Staubli VAL3: extAxisCan.pjx

--- extAxisCan.pjx ---
Parameters version=s7.6.3 stackSize=5000 millimeterUnit=true
Program file=CheckAxis.pgx
Program file=chkDrivesFault.pgx
Program file=chkDrivesOpEnab.pgx
Program file=chkDrivesSwOff.pgx
Program file=chkDrvState.pgx
Program file=chkLife.pgx
Program file=chkPosStatus.pgx
Program file=chkQuickStop.pgx
Program file=chkStatusWord.pgx
Program file=cmdAbortHoming.pgx
Program file=cmdDisableOp.pgx
Program file=cmdDisableVolt.pgx
Program file=cmdEnableHold.pgx
Program file=cmdEnableOp.pgx
Program file=cmdFaultReset.pgx
Program file=cmdQuickStop.pgx
Program file=cmdResetAll.pgx
Program file=cmdShutdown.pgx
Program file=cmdSwitchOn.pgx
Program file=getFbkPos.pgx
Program file=GoToPos.pgx
Program file=homing.pgx
Program file=init.pgx
Program file=IPMove.pgx
Program file=JogNegative.pgx
Program file=JogPositve.pgx
Program file=ReadMe.pgx
Program file=RecordExtAxis.pgx
Program file=RecordJoint.pgx
Program file=Reset.pgx
Program file=setCmdPos.pgx
Program file=setErrorCode.pgx
Program file=setHome.pgx
Program file=setOpMode.pgx
Program file=setPos.pgx
Program file=SingleMove.pgx
Program file=start.pgx
Program file=StepMove.pgx
Program file=stop.pgx
Program file=StopAll.pgx
Program file=stopExtAxis.pgx
Program file=Task4ms.pgx
Data file=extAxisCan.dtx
Library alias=cst path=Disk://constantes/constantes.pjx

--- extAxisCan.dtx ---
public aio aiPosFbk = {link=CanIO\Axis7\drvPosFbk_0}
public aio aoIPPos = {link=CanIO\Axis7\drvIPCmdPos_0}
public aio aoIPSpd = {link=CanIO\Axis7\ipVel_0}
public aio aoPosCmd = {link=CanIO\Axis7\drvCmdPos_0}
public aio aoWorkMode = {link=CanIO\Axis7\drvworkmode}
public bool bDriveQuickStop
public bool bDrivesOpEnable
bool bDrivesSwOnDis
public bool bDrvFault[2]
bool bEnableRequest
bool bIsS7_6 = true
bool bMemPower
public bool bNoDrivesFault = true
public bool bOpeEnabled[2]
bool bOverrun
public bool bQuickStop[2]
public bool bSWOnDis
public bool bSysShut
public bool blifebit[2]
  [0] = true
  [1] = true
bool blifebit_all_ok = true
public dio diFault = {link=CanIO\Axis7\fault_0}
public dio diHomingError = {link=CanIO\Axis7\homingError_0}
public dio diHomingReached = {link=CanIO\Axis7\homingReached_0}
public dio diIntLmtAct = {link=CanIO\Axis7\intLmtAct_0}
public dio diOpeEnabled = {link=CanIO\Axis7\opeEnabled_0}
public dio diPosReached = {link=CanIO\Axis7\targetReached_0}
public dio diQuickStop = {link=CanIO\Axis7\quickStopped_0}
public dio diReady2SwOn = {link=CanIO\Axis7\ready2SwOn_0}
public dio diSwOnDis = {link=CanIO\Axis7\swOnDis_0}
public dio diSwitchedOn = {link=CanIO\Axis7\switchedOn_0}
public dio diTargetReach = {link=CanIO\Axis7\targetReached_0}
public dio diVoltEnabled = {link=CanIO\Axis7\voltEnabled_0}
public dio diWarning = {link=CanIO\Axis7\warning_0}
public dio doEnableOp = {link=CanIO\Axis7\enableOp_0}
public dio doEnableVoltage = {link=CanIO\Axis7\enableVolt_0}
public dio doFaultReset = {link=CanIO\Axis7\faultReset_0}
public dio doManual = {link=CanIO\Axis7\Manual}
public dio doQuickStop = {link=CanIO\Axis7\quickStop_0}
public dio doStartHoming = {link=CanIO\Axis7\startHoming_0}
public dio doSwitchOn = {link=CanIO\Axis7\switchOn_0}
jointRx jDummy = {j1=1.48, j2=0.75, j3=2.04, j4=1.56, j5=2.81, j6=1.79}
jointRx jPosErrMax = {j1=100, j2=100, j3=100, j4=100, j5=100, j6=100}
jointRx jZero = {j1=0.01, j2=0.01, j3=0.01, j4=0.01, j5=0.01, j6=0.01}
public num nAxesPosFbk[2]
public num nAxesSum = 2
num nCntDrvDisable
num nCntDrvEnable[2]
public num nDrvFbkPos[2]
num nDrvPos[2]
num nDrvState[2]
  [0] = 1
  [1] = 1
public num nExtAxseAccDft = 10
public num nExtAxseSpdDft = 10
num nGearratio[2]
  [0] = 10
  [1] = 1
public num nResolution[2]
  [0] = 1280000
  [1] = 180000
public num nScaleFact[2]
  [0] = 10
  [1] = 360
public string sMsg
string sVersion = "s7.6 - May 29 2013 - 16:53:12"
public dio diRemote = {link=CanIO\Axis7\remote_0}
num nManul = 10
num nBuffSize
num nAxesData
public bool bMoveType
frame fFrame = {fatherId=world[0]}

--- start.pgx ---
program start()
  local num l_i
  local num l_sum
begin
  //
  call cst:init()
  call chkLife()
  if blifebit
    call init()
    taskCreateSync "T4ms",0.004,bOverrun,Task4ms()
  endIf
end

--- CheckAxis.pgx ---
public program CheckAxis(bool& x_b7Axis, bool& x_b8Axis)
begin

 x_b7Axis=$XgetNbAxes()>=1
 x_b8Axis=$XgetNbAxes()>=2


end

--- chkDrivesFault.pgx ---
program chkDrivesFault()
  local num l_i
begin
  //检查电机是否有错误
  //以下情况表明电机出现错误:
  //错误标志位；
  bNoDrivesFault=true
  for l_i=0 to nAxesSum-1
    if bDrvFault[l_i]!=(diFault[l_i]==true) and (!bDrvFault[l_i])
      sMsg="第"+toString("",l_i+1)+"轴控制器报错"
      popUpMsg(sMsg)
      logMsg(sMsg)
    endIf
    bDrvFault[l_i]=(diFault[l_i]==true)
    bNoDrivesFault=bNoDrivesFault and !bDrvFault[l_i]
  endFor
end

--- chkDrivesOpEnab.pgx ---
program chkDrivesOpEnab()
  local num l_i
begin
  //检查驱动器是否使能
  bDrivesOpEnable=true
  for l_i=0 to nAxesSum-1
    if  nDrvState[l_i]==5
      bOpeEnabled[l_i]=true
    else
      bOpeEnabled[l_i]=false
    endIf
    bDrivesOpEnable=bDrivesOpEnable and  bOpeEnabled[l_i]
  endFor

//
//  bDrivesOpEnable=bOpeEnabled[0]=(diOpeEnabled[0]==true and diSwitchedOn[0]==true and diQuickStop[0]==true )
//  for l_i=1 to nAxesSum-1
//    bOpeEnabled[l_i]=(diOpeEnabled[l_i]==true and diQuickStop[l_i]==true and  diSwitchedOn[l_i]==true )
//   // bOpeEnabled[l_i]=(diOpeEnabled[0]==true  and  diSwitchedOn[0]==true )
//    bDrivesOpEnable=bDrivesOpEnable and bOpeEnabled[l_i]
//  endFor
end

--- chkDrivesSwOff.pgx ---
program chkDrivesSwOff()
  local bool l_bDrvSwOnDis
  local num l_i
begin
  // 检测驱动器“switch on disabled"的状态
  bDrivesSwOnDis=true
  for l_i=0 to nAxesSum-1
    bSWOnDis[l_i]=(diSwOnDis[l_i]==true)
    bDrivesSwOnDis=bDrivesSwOnDis and bSWOnDis[l_i]
  endFor
  //
end

--- chkDrvState.pgx ---
program chkDrvState(num x_nAxisNum)
  local num l_nStatus
  local num l_nStatus1
  local bool l_bIsOneBitSet
begin
  //检查状态
  l_nStatus=0
  //确定电机是否在remote状态
  // read status_remote register
  //  call chkStatusRemote(x_nAxisNum,l_bIsOneBitSet)
  //  if l_bIsOneBitSet
  //    nDrvState[x_nAxisNum]=15
  //  else

  //读取状态字
  call chkStatusWord(x_nAxisNum,l_nStatus)
  //cst:nDRV_ACTIV:掩码，111dec=1101111bin.驱动器处于某种状态
  l_nStatus1=bAnd(l_nStatus,cst:nDRV_ACTIV)
  switch l_nStatus1
    //
    case cst:nRdy2SwitchON
      nDrvState[x_nAxisNum]=3
    break
    //
    case cst:nSwitchedON
      nDrvState[x_nAxisNum]=4
    break
    //使能
    case cst:nOperatEnabled
      nDrvState[x_nAxisNum]=5
    break
    //quickstop
    case cst:nQuickStopActiv
      nDrvState[x_nAxisNum]=12
    break
    //
    default
      //cst:nDRV_FAULT=100 1111
      l_nStatus1=bAnd(l_nStatus,cst:nDRV_FAULT)

      switch l_nStatus1
        case cst:nNotRdySwiON
          nDrvState[x_nAxisNum]=1
        break
        //
        case cst:nSwitchONDis
          nDrvState[x_nAxisNum]=2
        break
        //
        case cst:nFaultReacActiv
          nDrvState[x_nAxisNum]=13
        break
        //
        case cst:nFaultState
          nDrvState[x_nAxisNum]=14
        break
        //
        default
          nDrvState[x_nAxisNum]=-1
        break
      endSwitch
    break
    //
  endSwitch
end

--- chkLife.pgx ---
public program chkLife()
  local num l_i
  local string l_sMsg
begin
  //检查IO连接是否正常
  blifebit_all_ok=true
  for l_i=0 to nAxesSum-1
    if ioStatus(diReady2SwOn[l_i])<0
      blifebit[l_i]=false
      l_sMsg="第"+toString("",l_i+1)+"轴通讯异常"
      popUpMsg(l_sMsg)
      logMsg(l_sMsg)
      blifebit_all_ok=blifebit_all_ok and blifebit[l_i]
      return
    else
      blifebit[l_i]=true
      blifebit_all_ok=blifebit_all_ok and blifebit[l_i]
    endIf
  endFor

end

--- chkPosStatus.pgx ---
public program chkPosStatus(bool& x_bIsSame, num x_nAxisNum, num x_nAxisPos)
begin
  //检查外部轴是否在指定位置上
  x_bIsSame=abs(aioGet(aiPosFbk[x_nAxisNum])-x_nAxisPos*nGearratio[x_nAxisNum]*nResolution[x_nAxisNum]/nScaleFact[x_nAxisNum])<=5
end

--- chkQuickStop.pgx ---
program chkQuickStop()
  local num l_ni
begin
  //
  bDriveQuickStop=false
  for l_ni=0 to nAxesSum-1
    if nDrvState[l_ni]==12
      bQuickStop[l_ni]=true
    else
      bQuickStop[l_ni]=false
    endIf
    bDriveQuickStop=bDriveQuickStop or bQuickStop[l_ni]
  endFor
end

--- chkStatusWord.pgx ---
program chkStatusWord(num x_nAxisNumber, num& x_nValue)
begin
  //返回电机状态字的数值
  //  x_nValue=aioGet(aiStatusWord[x_nAxisNumber])
  x_nValue=dioGet(diReady2SwOn[x_nAxisNumber])*power(2,0)
  x_nValue=dioGet(diSwitchedOn[x_nAxisNumber])*power(2,1)+x_nValue
  x_nValue=dioGet(diOpeEnabled[x_nAxisNumber])*power(2,2)+x_nValue
  x_nValue=dioGet(diFault[x_nAxisNumber])*power(2,3)+x_nValue
  x_nValue=dioGet(diVoltEnabled[x_nAxisNumber])*power(2,4)+x_nValue
  x_nValue=dioGet(diQuickStop[x_nAxisNumber])*power(2,5)+x_nValue
  x_nValue=dioGet(diSwOnDis[x_nAxisNumber])*power(2,6)+x_nValue
  x_nValue=dioGet(diWarning[x_nAxisNumber])*power(2,7)+x_nValue
  x_nValue=dioGet(diRemote[x_nAxisNumber])*power(2,9)+x_nValue
  x_nValue=dioGet(diTargetReach[x_nAxisNumber])*power(2,10)+x_nValue
  x_nValue=dioGet(diIntLmtAct[x_nAxisNumber])*power(2,11)+x_nValue
  x_nValue=dioGet(diHomingReached[x_nAxisNumber])*power(2,12)+x_nValue
  x_nValue=dioGet(diHomingError[x_nAxisNumber])*power(2,13)+x_nValue
end

--- cmdAbortHoming.pgx ---
public program cmdAbortHoming(num x_nAxisNum)
begin
 //取消回零

end

--- cmdDisableOp.pgx ---
public program cmdDisableOp(num x_nAxNum)
begin
  //发送“终止操作”指令到所选驱动器
  if bOpeEnabled[x_nAxNum]==true
    doFaultReset[x_nAxNum]=false
    doEnableOp[x_nAxNum]=false
    delay(0.1)
    doQuickStop[x_nAxNum]=true
    doEnableVoltage[x_nAxNum]=true
    doSwitchOn[x_nAxNum]=true
  endIf
end

--- cmdDisableVolt.pgx ---
public program cmdDisableVolt(num x_nAxNum)
begin
  //"Disable voltage"字段无效
  doFaultReset[x_nAxNum]=false
  doEnableVoltage[x_nAxNum]=false
end

--- cmdEnableHold.pgx ---
public program cmdEnableHold(num x_nAxNum (dimensions=1))
begin
  // this program issues an 'Enable Hold'  command to the selected drive.
  // This bit must be set to enable drive power
  //发送“enable hold”指令到所选控制器
  //用于设置驱动器电源开启
  //  doEnableHold[x_nAxNum]=true
end

--- cmdEnableOp.pgx ---
public program cmdEnableOp(num x_nAxNum)
begin
  //设置'Enable Operation'
  if bOpeEnabled[x_nAxNum]==false
    doFaultReset[x_nAxNum]=false
    doSwitchOn[x_nAxNum]=false
    doEnableOp[x_nAxNum]=false
    doEnableVoltage[x_nAxNum]=true
    doQuickStop[x_nAxNum]=true
    delay(0.1)
    doSwitchOn[x_nAxNum]=true
    delay(0.1)
    doEnableOp[x_nAxNum]=true
    delay(0.1)
  endIf
end

--- cmdFaultReset.pgx ---
public program cmdFaultReset(num x_nAxNum)
begin
  //错误复位，'Fault reset'置1
  doFaultReset[x_nAxNum]=true
  delay(0.008)
  doFaultReset[x_nAxNum]=false
end

--- cmdQuickStop.pgx ---
public program cmdQuickStop(num x_nAxNum)
begin
  //"quickstop"置为false
  //激活quickstop
  if !bQuickStop[x_nAxNum]
    doFaultReset[x_nAxNum]=false
    doEnableVoltage[x_nAxNum]=true
    doSwitchOn[x_nAxNum]=true
    doEnableOp[x_nAxNum]=true
    delay(0.1)
    doQuickStop[x_nAxNum]=false
    delay(0.1)
  endIf
end

--- cmdResetAll.pgx ---
public program cmdResetAll(num x_nAxNum)
begin
  //复位所有信号
  doFaultReset[x_nAxNum]=false
  doEnableOp[x_nAxNum]=false
  doSwitchOn[x_nAxNum]=false
  doEnableVoltage[x_nAxNum]=false
  doQuickStop[x_nAxNum]=false
  delay(0.1)
end

--- cmdShutdown.pgx ---
public program cmdShutdown(num& x_nAxNum)
begin
  //关闭指定驱动器，设置"switch on"为false
  //shutdown的顺序参考相应电机说明
  doFaultReset[x_nAxNum]=false
  doQuickStop[x_nAxNum]=true
  doEnableVoltage[x_nAxNum]=true
  doSwitchOn[x_nAxNum]=false
  delay(0.004)
end

--- cmdSwitchOn.pgx ---
public program cmdSwitchOn(num& x_nAxNum)
begin
  //"switch on"设置为true
  doFaultReset[x_nAxNum]=false
  doEnableOp[x_nAxNum]=false
  doQuickStop[x_nAxNum]=true
  doEnableVoltage[x_nAxNum]=true
  doSwitchOn[x_nAxNum]=true
  delay(0.1)
end

--- DAEMON1.PGX ---
public program daemon1()
  local num l_nKey
begin

  while (getKey()!=270)
    call daemon4()
    delay(0)
  endWhile
end

--- DAEMON2.PGX ---
public program daemon2()
  local jointRx l_jCurr
  local num l_i
  local bool l_bError
  local string l_sMsg
  local num l_nError
  local bool l_bDrivesOK
begin

  // Verification du bit de vie bus can
  call chkLifeBit()

  // Gestion watchDog pour variateurs
  //call updateWatchDog()
  //
  // Recupere etat des variateurs
  l_bDrivesOK=true
  for l_i=0 to nNUMOFAXES-1
    bDrvFault[l_i]=(diFault[l_i]==true) or bAnd(aioGet(aiStatusRemote[l_i])/32,255)!=0
    call chkDrvState(l_i)
    l_bDrivesOK=l_bDrivesOK and nDrvState[l_i]==cst:nOperatEnabled
    bDrivesOpEnable=l_bDrivesOK
  endFor

  if isPowered() and l_bDrivesOK
    // Get system position
    $XgetDrvCmdPos(nDrvPos)
    l_sMsg=""
    //$XgetJntCmdPos(l_nJntPos)
    for l_i=0 to nNUMOFAXES-1
      // Send it to the external axis
      aioSet(aoPosCmd[l_i],nDrvPos[l_i]*nScaleFact)
      //l_sMsg="0: "+toString(".3",l_nJntPos[0])+"   1: "+toString(".3",l_nJntPos[1])
      l_sMsg=l_sMsg+toString("",l_i)+": "+toString(".3",nDrvPos[l_i])+"   "
    endFor
    //? l_sMsg
  else
    for l_i=0 to nNUMOFAXES-1
      doEnableOp[l_i]=false
      doSwitchOn[l_i]=false
      // Get external axis position
      nDrvPos[l_i]=aioGet(aiPosFbk[l_i])/nScaleFact
    endFor
    // Update it in the system
    $XsetDrvFbkPos(nDrvPos)
  endIf



end

--- getFbkPos.pgx ---
public program getFbkPos()
  local num l_i
begin
  for l_i=0 to nAxesSum-1
      //nScaleFact:电机转一圈角度（旋转轴）或前进距离（直线轴（mm））
      nDrvFbkPos[l_i]=nScaleFact[l_i]*aioGet(aiPosFbk[l_i])/nResolution[l_i]*nGearratio[l_i]
      nAxesPosFbk[l_i]=nDrvFbkPos[l_i]/nGearratio[l_i]
  endFor
end

--- getStatusWord.pgx ---
public program getStatusWord(num x_nAxisNumber, num& x_nValue)
begin
  // this routine return the value of the drive's status word
  //
  x_nValue=aioGet(aiStatusWord[x_nAxisNumber])
end

--- GoToPos.pgx ---
public program GoToPos(num x_nAxisNum, num x_nPos)
begin

  if !isPowered()
    popUpMsg("请先给机器人上电")
    return
  endIf
  doStartHoming[x_nAxisNum]=false
  aioSet(aoWorkMode[x_nAxisNum],cst:nPPMODE)
  delay(0.1)
  aioSet(aoPosCmd[x_nAxisNum],x_nPos*nResolution[x_nAxisNum]/nScaleFact[x_nAxisNum])
  delay(0.1)
  doStartHoming[x_nAxisNum]=true
  doManual[x_nAxisNum]=true
  wait(diTargetReach[x_nAxisNum]==false)
  wait(diTargetReach[x_nAxisNum]==true)
  disablePower()
  delay(0.1)
  aioSet(aoWorkMode[x_nAxisNum],cst:nINTERPMODE)
  doStartHoming[x_nAxisNum]=true
end

--- homing.pgx ---
public program homing(num x_nAxisNum, bool& x_bRes)
  local bool l_bError
  local num l_nEtape
  local string l_sMsg
  local num l_nTps
  local bool l_bVerrou
  local bool l_bOK
  local num l_nDuration
  local string l_sYN[2]
  local num l_nDrvPos
begin
  //指定外部轴零点
  //  if !isPowered()
  //    popUpMsg("请先上电")
  //    return
  //  endIf
  //  x_bRes=false
  //  doStartHoming[x_nAxisNum]=false
  //  delay(0.1)
  //  aioSet(aoWorkMode[x_nAxisNum],6)
  //  doStartHoming[x_nAxisNum]=true
  //  l_sYN[0]="是"
  //  l_sYN[1]="否"
  //  if watch(diHomingReached[x_nAxisNum]==true,2)
  //    x_bRes=true
  //    popUpMsg("设置成功")
  //  endIf

  //
  x_bRes=false
  if !isPowered()
    popUpMsg("请先给机器人上电")
    return
  endIf
  doStartHoming[x_nAxisNum]=false
  aioSet(aoWorkMode[x_nAxisNum],cst:nHOMINGMODE)
  delay(0.1)
  doStartHoming[x_nAxisNum]=true
  wait(diHomingReached[x_nAxisNum]==false)
  wait(diHomingReached[x_nAxisNum]==true)
  disablePower()
  delay(0.1)
  aioSet(aoWorkMode[x_nAxisNum],cst:nINTERPMODE)
  x_bRes=true
end

--- init.pgx ---
public program init()
  local num l_i
  local bool l_bError
begin

  call cst:init()
  //获取外部轴数目
  nAxesSum=$XgetNbAxes()

  if nAxesSum<1
    popUpMsg("外部轴不正确")
    return
  endIf

  //根据外部轴数目更改变量数目
  resize(nCntDrvEnable,1,nAxesSum)
  resize(nDrvPos,1,nAxesSum)
  resize(bDrvFault,1,nAxesSum)
  resize(nAxesPosFbk,1,nAxesSum)
  resize(nDrvFbkPos,1,nAxesSum)
  resize(bDrvFault,1,nAxesSum)
  resize(bOpeEnabled,1,nAxesSum)
  resize(bQuickStop,1,nAxesSum)
  resize(blifebit,1,nAxesSum)
  resize(nDrvState,1,nAxesSum)
  //  if size(nDrvPos)!=nAxesSum
  //    resize(nDrvPos,1,nAxesSum)
  //  endIf

  //  if size(nDrvFbkPos)!=nAxesSum
  //    resize(nDrvFbkPos,1,nAxesSum)
  //  endIf
  //  if size(bDrvFault)!=nAxesSum
  //    resize(bDrvFault,1,nAxesSum)
  //  endIf
  //  if size(nAxesPosFbk)!=nAxesSum
  //    resize(nAxesPosFbk,1,nAxesSum)
  //  endIf
  //  if size(bOpeEnabled)!=nAxesSum
  //    resize(bOpeEnabled,1,nAxesSum)
  //  endIf
  //
  //  if size(bQuickStop)!=nAxesSum
  //    resize(bQuickStop,1,nAxesSum)
  //  endIf
  //
  //  if size(blifebit)!=nAxesSum
  //    resize(blifebit,1,nAxesSum)
  //  endIf
  //
  //  if size(nCntDrvEnable)!=nAxesSum
  //    resize(nCntDrvEnable,1,nAxesSum)
  //  endIf
  //
  //  // 驱动器状态变量
  //  if size(nDrvState)!=nAxesSum
  //    resize(nDrvState,1,nAxesSum)
  //  endIf
  //
  //





  //初始化
  for l_i=0 to nAxesSum-1
    call cmdResetAll(l_i)
    call cmdFaultReset(l_i)
    bDrvFault[l_i]=false
    aioSet(aoWorkMode[l_i],cst:nINTERPMODE)
    doStartHoming[l_i]=true
    nCntDrvEnable[l_i]=0
    bQuickStop=false
  endFor
  delay(0.008)
  disablePower()
  wait(isPowered()==false)
  bSysShut=false
  //
  // call Version()
  // libSave()
end

--- IPMove.pgx ---
public program IPMove()
begin
  //
//  $XgetDrvCmdPos(nDrvPos)
//  for l_i=0 to nAxesSum-1
//    aioSet(aoIPPos[l_i],(nDrvPos[l_i]*nResolution[l_i]/nScaleFact[l_i]))
//  endFor
end

--- JogNegative.pgx ---
public program JogNegative(num x_nAxis, num x_nKey)
begin
  call StepMove(x_nAxis,x_nKey,false)
end

--- JogPositve.pgx ---
public program JogPositve(num x_nAxis, num x_nKey)
begin
  call StepMove(x_nAxis,x_nKey,true)
end

--- pwrOffDrive1.pgx ---
public program pwrOffDrive1(num x_nAxNum, num& x_nError)
  local bool l_bVerrou
  local num l_nEtape
  local bool l_bOK
  local string l_sMsg
  local num l_nMemEtape
  local bool l_bQuit
begin

  l_bVerrou=false
  l_nMemEtape=-1
  l_bQuit=false
  x_nError=0

  // sequenceur pour desactiver les variateurs
  while !l_bQuit
    // Read current drive State
    //call getDriveState(x_nAxNum,nDrvState[x_nAxNum])
    l_nEtape=nDrvState[x_nAxNum]
    // Changement d'état ?
    if l_nEtape!=l_nMemEtape
      l_nMemEtape=l_nEtape
      l_bVerrou=false
    endIf

    l_sMsg="pwrOffDrive>>Etape : "+toString("",l_nEtape)+" "
    switch l_nEtape
      // Not ready to Switch on
      case 1
        if l_bVerrou==false
          if bAnd(nDebug,cst:nDEBUGDRIVE)==cst:nDEBUGDRIVE
            l_sMsg=l_sMsg+"Not ready to Switch on"
            logMsg(l_sMsg)
          endIf
          l_bVerrou=true
        endIf
      break
      // Switch ON disabled
      case 2
        if l_bVerrou==false
          if bAnd(nDebug,cst:nDEBUGDRIVE)==cst:nDEBUGDRIVE
            l_sMsg=l_sMsg+"Switch on disabled"
            logMsg(l_sMsg)
          endIf
          l_bQuit=true
          call cmdResetAll(x_nAxNum)
          l_bVerrou=true
        endIf
      break
      // Ready to switch on
      case 3
        if l_bVerrou==false
          if bAnd(nDebug,cst:nDEBUGDRIVE)==cst:nDEBUGDRIVE
            l_sMsg=l_sMsg+"Ready to switch on"
            logMsg(l_sMsg)
          endIf
          call cmdQuickStop(x_nAxNum)
          call cmdDisableVolt(x_nAxNum)
          l_bVerrou=true
        endIf
      break
      // Switched ON
      case 4
        if l_bVerrou==false
          if bAnd(nDebug,cst:nDEBUGDRIVE)==cst:nDEBUGDRIVE
            l_sMsg=l_sMsg+"Switched ON"
            logMsg(l_sMsg)
          endIf
          //          call cmdQuickStop(x_nAxNum)
          //          call cmdDisableVolt(x_nAxNum)
          //
          call cmdShutdown(x_nAxNum)
          l_bVerrou=true
        endIf
      break
      // Operation enabled
      case 5
        if l_bVerrou==false
          if bAnd(nDebug,cst:nDEBUGDRIVE)==cst:nDEBUGDRIVE
            l_sMsg=l_sMsg+"Operation enabled"
            logMsg(l_sMsg)
          endIf
          //          call cmdDisableVolt(x_nAxNum)

          //*******
          call cmdDisableOp(x_nAxNum)
          // ******
          l_bVerrou=true
        endIf
      break

      // Fault state
      case 14
        if l_bVerrou==false
          if bAnd(nDebug,cst:nDEBUGDRIVE)==cst:nDEBUGDRIVE
            l_sMsg=l_sMsg+"Fault state"
            logMsg(l_sMsg)
          endIf
          l_bQuit=true
          x_nError=1
          l_bVerrou=true
        endIf
      break
      //
      // Alarm from status_remote register is set
      case 15
        if l_bVerrou==false
          if bAnd(nDebug,cst:nDEBUGDRIVE)==cst:nDEBUGDRIVE
            l_sMsg=l_sMsg+"Alarm Status_remote register"
            logMsg(l_sMsg)
          endIf
          l_bQuit=true
          x_nError=2
          call cmdResetAll(x_nAxNum)
          l_bVerrou=true
        endIf
      break
      //
    endSwitch
    delay(0)
  endWhile

end

--- pwrOffDrive2.pgx ---
public program pwrOffDrive2(num x_nAxNum)
  local bool l_bOK
  local string l_sMsg
begin
  // sequenceur pour desactiver les variateurs

  // Read current drive State
  call chkDrvState(x_nAxNum)

  // Changement d'état ?
  if nDrvState[x_nAxNum]!=nMemPwrOffStep[x_nAxNum]
    nMemPwrOffStep[x_nAxNum]=nDrvState[x_nAxNum]
    bLockPwrOff[x_nAxNum]=false
  endIf

  l_sMsg="pwrOffDrive>>Etape : "+toString("",nDrvState[x_nAxNum])+" "
  switch nDrvState[x_nAxNum]
    // Not ready to Switch on
    case 1
      if bLockPwrOff[x_nAxNum]==false
        if bAnd(nDebug,cst:nDEBUGDRIVE)==cst:nDEBUGDRIVE
          l_sMsg=l_sMsg+"Not ready to Switch on"
          logMsg(l_sMsg)
        endIf
        bLockPwrOff[x_nAxNum]=true
      endIf
    break
    // Switch ON disabled
    case 2
      if bLockPwrOff[x_nAxNum]==false
        if bAnd(nDebug,cst:nDEBUGDRIVE)==cst:nDEBUGDRIVE
          l_sMsg=l_sMsg+"Switch on disabled"
          logMsg(l_sMsg)
        endIf
        call cmdResetAll(x_nAxNum)
        bLockPwrOff[x_nAxNum]=true
      endIf
    break
    // Ready to switch on
    case 3
      if bLockPwrOff[x_nAxNum]==false
        if bAnd(nDebug,cst:nDEBUGDRIVE)==cst:nDEBUGDRIVE
          l_sMsg=l_sMsg+"Ready to switch on"
          logMsg(l_sMsg)
        endIf
        call cmdQuickStop(x_nAxNum)
        call cmdDisableVolt(x_nAxNum)
        bLockPwrOff[x_nAxNum]=true
      endIf
    break
    // Switched ON
    case 4
      if bLockPwrOff[x_nAxNum]==false
        if bAnd(nDebug,cst:nDEBUGDRIVE)==cst:nDEBUGDRIVE
          l_sMsg=l_sMsg+"Switched ON"
          logMsg(l_sMsg)
        endIf
        call cmdShutdown(x_nAxNum)
        bLockPwrOff[x_nAxNum]=true
      endIf
    break
    // Operation enabled
    case 5
      if bLockPwrOff[x_nAxNum]==false
        if bAnd(nDebug,cst:nDEBUGDRIVE)==cst:nDEBUGDRIVE
          l_sMsg=l_sMsg+"Operation enabled"
          logMsg(l_sMsg)
        endIf
        call cmdDisableOp(x_nAxNum)
        bLockPwrOff[x_nAxNum]=true
      endIf
    break

    // Fault state
    case 14
      if bLockPwrOff[x_nAxNum]==false
        if bAnd(nDebug,cst:nDEBUGDRIVE)==cst:nDEBUGDRIVE
          l_sMsg=l_sMsg+"Fault state"
          logMsg(l_sMsg)
        endIf
        bLockPwrOff[x_nAxNum]=true
      endIf
    break
    //
    // Alarm from status_remote register is set
    case 15
      if bLockPwrOff[x_nAxNum]==false
        if bAnd(nDebug,cst:nDEBUGDRIVE)==cst:nDEBUGDRIVE
          l_sMsg=l_sMsg+"Alarm Status_remote register"
          logMsg(l_sMsg)
        endIf
        call cmdResetAll(x_nAxNum)
        bLockPwrOff[x_nAxNum]=true
      endIf
    break
    //
  endSwitch

end

--- pwrOffDrives.pgx ---
public program pwrOffDrives()
  local num l_i
begin
  for l_i=0 to nNUMOFAXES-1
    doEnableVoltage[l_i]=false
    doQuickStop[l_i]=false
    doSwitchOn[l_i]=false
    doEnableOp[l_i]=false
  endFor
end

--- ReadMe.pgx ---
program ReadMe()
begin
//在通用版本上对lasman进行定制
//1.添加了三个四个函数
//checkAxis
//SingleMove
//RecordExtAxis
//RecordJoint


//还有一些变量需要添加







end

--- RecordExtAxis.pgx ---
public program RecordExtAxis(trsf& x_trTrsf, trsf& x_trPos, tool x_tTool)
  local jointRx l_jJ
  local pointRx l_pP
begin
  //  $recClean("c")
  //  $recAdd("c","CanIO\Axis8\posCmd_1")
  //  $recAdd("c","CanIO\Axis8\posFbk_1")
  //  $recStart("c",50,250)

  //  $recClean("c")
  //  $recAdd("c","extDrvCmdPos")
  //  $recAdd("c","extDrvCmdVel")
  //  $recAdd("c","extJntCmdPos")
  //  $recAdd("c","extJntCmdVel")
  //  $recAdd("c","extError")
  //  $recAdd("c","extDrvGrpError")
  //  $recStart("c",50,250)

 // x_pPos=$here
//    resize(nBuffSize,1,sel(x_b8Axis,2,1))
//  x_j=$XH(nBuffSize)
//  x_trTrsf.x=nBuffSize[0]
//  if x_b8Axis
//    x_trTrsf.y=nBuffSize[1]
//  endIf


if bMoveType
  $XframeLink(fFrame)
 l_pP=here(x_tTool,fFrame)
  x_trPos=l_pP.trsf

endIf




//记录七轴，八轴位置
call RecordJoint(l_jJ,x_trTrsf)




end

--- RecordJoint.pgx ---
public program RecordJoint(jointRx& x_j, trsf& x_trTrsf)
  local num l_nNum[2]
begin
  //  $recClean("c")
  //  $recAdd("c","CanIO\Axis8\posCmd_1")
  //  $recAdd("c","CanIO\Axis8\posFbk_1")
  //  $recStart("c",50,250)

  //  $recClean("c")
  //  $recAdd("c","extDrvCmdPos")
  //  $recAdd("c","extDrvCmdVel")
  //  $recAdd("c","extJntCmdPos")
  //  $recAdd("c","extJntCmdVel")
  //  $recAdd("c","extError")
  //  $recAdd("c","extDrvGrpError")
  //  $recStart("c",50,250)

 // x_pPos=$here

 //记录轴的值
  if nAxesSum<1
    popUpMsg("轴个数错误")
    return
  endIf

  resize(nBuffSize,1,nAxesSum)
  x_j=$Xherej(nBuffSize)
  x_trTrsf.x=nBuffSize[0]
  if nAxesSum>1
    x_trTrsf.y=nBuffSize[1]
  endIf

end

--- Reset.pgx ---
public program Reset()
  local num l_i
begin
  //报警复位
  for l_i=0 to nAxesSum-1
    call cmdFaultReset(l_i)
  endFor
//  call user:timerDialog("复位完成",0.5)
end

--- setCmdPos.pgx ---
program setCmdPos(num x_nAxisNum (dimensions=1))
  local num l_nCurrentPos
  local num l_nCmdPos
begin
  //把当前位置赋给驱动器
  l_nCurrentPos=aioGet(aiPosFbk[x_nAxisNum])
  aioSet(aoPosCmd[x_nAxisNum],l_nCurrentPos)
end

--- setErrorCode.pgx ---
program setErrorCode(num x_nAxisNum (dimensions=1), num& x_nErrorCode (dimensions=1))
  local num l_nAlarm
begin
  // This program returns the value of the current error
  //获取当前错误代码值
  x_nErrorCode=0
  //检查电机错误位是否被设置
  // Check if driveFault bit is set
  //  if diFault[x_nAxisNum]==true
  //    //硬件错误
  //    // Hardware alarm ?
  //    call chkHwAlarm(x_nAxisNum,x_nErrorCode)
  //    if x_nErrorCode==0
  //      // Software alarm ?
  //      call chkSwAlarm(x_nAxisNum,x_nErrorCode)
  //    endIf
  //    // Check alarm bits of status_remote register
  //  elseIf nAppV3Error[x_nAxisNum]==0
  //    call getRegisterVal(cst:nSTATUS_REMOTE,x_nAxisNum,x_nErrorCode)
  //  else
  //    // Check if Application error
  //    x_nErrorCode=nAppV3Error[x_nAxisNum]
  //  endIf
end

--- setHome.pgx ---
public program setHome(num x_nAxisNum, bool& x_bRes)
  local bool l_bError
  local num l_nEtape
  local string l_sMsg
  local num l_nTps
  local bool l_bVerrou
  local bool l_bOK
  local num l_nDuration
  local string l_sYN[2]
  local num l_nDrvPos
begin
  //对绝对编码器电机设置当前值位为零点
    if !isPowered()
      popUpMsg("请先上电")
      return
    endIf
    x_bRes=false
    doStartHoming[x_nAxisNum]=false
    delay(0.1)
    aioSet(aoWorkMode[x_nAxisNum],cst:nHOMINGMODE)
    doStartHoming[x_nAxisNum]=true
    wait(diHomingReached[x_nAxisNum]==false)
    wait(diHomingReached[x_nAxisNum]==true)
    if watch(diHomingReached[x_nAxisNum]==true,2)
      x_bRes=true
      popUpMsg("设置成功")
    endIf
    disablePower()
    delay(0.008)
    aioSet(aoWorkMode[x_nAxisNum],cst:nINTERPMODE)
 end

--- setOpMode.pgx ---
public program setOpMode(num x_nAxisNum, num x_nOpMode)
  local num l_nK
begin

  //call checkDin(diSwitchedOn[x_nAxisNum],false,x_bError)

  // Interpolated position mode
  //  aioSet(aoMoop[x_nAxisNum],x_nOpMode)
  aioSet(aoWorkMode[x_nAxisNum],x_nOpMode)
  // Reset fault
//  doFaultReset[x_nAxisNum]=false
//  delay(0.1)
//  doFaultReset[x_nAxisNum]=true
//  delay(0.1)
//  doFaultReset[x_nAxisNum]=false

  // Copy current axis position into commanded position
  // Probably not necessary need to be checked.
  //  call setCmdPos(x_nAxisNum)

  //  // Init watchdog
  //  doEnableHold[x_nAxisNum]=true
  //  doWatchDog[x_nAxisNum]=true
  //  // Starting sequence
  //  doEnableVoltage[x_nAxisNum]=true
  //  doQuickStop[x_nAxisNum]=true

  //call checkDin(diReady2SwOn[x_nAxisNum],true,x_bError)


end

--- setPos.pgx ---
program setPos(num x_nAxisNum (dimensions=1), num x_nCurrentPos (dimensions=1))
begin
  //
  aioSet(aoPosCmd[x_nAxisNum],x_nCurrentPos)
end

--- SingleMove.pgx ---
public program SingleMove(num x_nType, jointRx x_j, pointRx x_pM, pointRx x_pE, tool x_tTool, mdesc x_m, trsf x_trExtAxis)
  local pointRx l_pP[2]
begin
  if x_nType<1 or x_nType>3
    return
  endIf

  resize(nAxesData,1,nAxesSum)
  nAxesData[0]=x_trExtAxis.x
  if nAxesSum>=2
    nAxesData[1]=x_trExtAxis.y

  endIf



  if !bMoveType or x_nType==1

    switch x_nType
      case 1
        $Xmovej(x_j,nAxesData,x_tTool,x_m)
      break


      case 2
        $Xmovel(x_pE,nAxesData,x_tTool,x_m)
      break

      case 3
        $Xmovec(x_pM,x_pE,nAxesData,x_tTool,x_m)
      break


    endSwitch
    return


  endIf





  //2014.12.04
  //对于离线进行修改
  //fFrame.trsf={0,0,0,0,0,0}
  if bMoveType
    $XframeLink(fFrame)
  else
    link(fFrame,world)
  endIf





  link(l_pP[0],fFrame)
  link(l_pP[1],fFrame)


  l_pP[0].trsf=x_pM.trsf
  l_pP[1].trsf=x_pE.trsf

  //×××××××××××××××××××××××××××××××××××××××××××
  switch x_nType
    case 1
      $Xmovej(x_j,nAxesData,x_tTool,x_m)
    break

    case 2
      $Xmovel(l_pP[1],nAxesData,x_tTool,x_m)
    break

    case 3
      $Xmovec(l_pP[0],l_pP[1],nAxesData,x_tTool,x_m)
    break

  endSwitch


end

--- StepMove.pgx ---
public program StepMove(num x_nAxisNum, num x_nKey, bool x_bJog)
begin
  //
  if isKeyPressed(x_nKey)
    //x_bjog=true:正向运动
    if x_bJog
      ? "+"
      aioSet(aoWorkMode[x_nAxisNum],-1)
      doStartHoming[x_nAxisNum]=true
    else
      ? "-"
      aioSet(aoWorkMode[x_nAxisNum],-1)
      doManual[x_nAxisNum]=true
    endIf
    wait(isKeyPressed(x_nKey)==false)
  else
    doStartHoming[x_nAxisNum]=false
    doManual[x_nAxisNum]=false
  endIf
end

--- stop.pgx ---
public program stop()
  local num l_i
begin
  call StopAll()


end

--- StopAll.pgx ---
public program StopAll()
  local num l_ni
begin
  for l_ni=0 to nAxesSum-1
    call stopExtAxis(l_ni)
  endFor
end

--- stopExtAxis.pgx ---
public program stopExtAxis(num x_nAxisNum)
begin
  //
  if blifebit[x_nAxisNum]
    doQuickStop[x_nAxisNum]=false
    doSwitchOn[x_nAxisNum]=false
    doEnableVoltage[x_nAxisNum]=false
    doEnableOp[x_nAxisNum]=false
    doStartHoming[x_nAxisNum]=false
    aioSet(aoWorkMode[x_nAxisNum],0)
  endIf
end

--- SYNCMOVE.pgx ---
public program syncMove(num& x_nAxisNum[])
  local jointRx l_jCurr
  local num l_nEncRes
  local num l_nDrvPos[2]
  local bool l_bFirstRun
  local num l_i
  local bool l_bError
  local string l_sMsg
begin

  l_nEncRes=8192/360

  call setCmdPos(0)
  call setCmdPos(1)
  bStop=false
  l_bFirstRun=true

  // Ne pas supprimer ces lignes
  disablePower()
  wait(isPowered()==false)
  //wait(isPowered()==true)
  /// FIN /////////////

  while !bStop
    if (isPowered()==true) and (l_bFirstRun==false)
      for l_i=0 to size(x_nAxisNum)-1
        if (diSwitchedOn[x_nAxisNum[l_i]]==false)
          doSwitchOn[x_nAxisNum[l_i]]=true
          delay(0.05)
          doEnableOp[x_nAxisNum[l_i]]=true
        endIf
      endFor
      // Get system position
      $XgetDrvCmdPos(l_nDrvPos)
      //$XgetJntCmdPos(l_nJntPos)
      // Send it to the external axis
      aioSet(aoPosCmd[x_nAxisNum[0]],l_nDrvPos[0]*l_nEncRes)
      aioSet(aoPosCmd[x_nAxisNum[1]],l_nDrvPos[1]*l_nEncRes)
      //l_sMsg="0: "+toString(".3",l_nJntPos[0])+"   1: "+toString(".3",l_nJntPos[1])
      l_sMsg="0: "+toString(".3",l_nDrvPos[0])+"   1: "+toString(".3",l_nDrvPos[1])
      //? l_sMsg
    else
      for l_i=0 to size(x_nAxisNum)-1
        doSwitchOn[x_nAxisNum[l_i]]=false
        doEnableOp[x_nAxisNum[l_i]]=false
      endFor
      // Get external axis position
      l_nDrvPos[0]=aioGet(aiPosFbk[x_nAxisNum[0]])/l_nEncRes
      l_nDrvPos[1]=aioGet(aiPosFbk[x_nAxisNum[1]])/l_nEncRes
      // Update it in the system
      $XsetDrvFbkPos(l_nDrvPos)
    endIf
    delay(0)
    l_bFirstRun=false
  endWhile
end

--- Task4ms.pgx ---
public program Task4ms()
  local num l_i
  local num l_nWorking
  local num l_nStatus
begin
  //4ms的任务,检测外部轴的状态信息
  while true
    //检查通讯是否正常
    call chkLife()
    if !blifebit_all_ok
      resetMotion()
      stopMove()
      disablePower()
      popUpMsg("同步外部轴异常")
      bSysShut=true
      return
    endIf
    //检查错误
    call chkDrivesFault()
    //检查状态
    for l_i=0 to nAxesSum-1
      call chkDrvState(l_i)
    endFor
    //反馈位置
    call getFbkPos()
    // 检查所有驱动器是否在operation enabled
    call chkDrivesOpEnab()
    //检测quickstop
    call chkQuickStop()
    //s7.6以上版本


    //使用在s7.5及以下系统时，命令行注释
    bEnableRequest=isPowered()
    //使用在s7.6，命令行注释
    $XdrvEnable(bEnableRequest,bDrivesOpEnable)
    //
    if bEnableRequest
      if bMemPower==false
        // 触发使能次数
        for l_i=0 to nAxesSum-1
          nCntDrvEnable[l_i]=0
        endFor
        bMemPower=true
      endIf
      //
      if bNoDrivesFault
        if bDrivesOpEnable
          //从$XMovel,$XMovej和$XMovec指令中获得外部轴离散位置(4ms的距离)
          $XgetDrvCmdPos(nDrvPos)
          for l_i=0 to nAxesSum-1
            aioSet(aoIPPos[l_i],(nDrvPos[l_i]/nGearratio[l_i]*nResolution[l_i]/nScaleFact[l_i]))
          endFor
          bSysShut=false
        else
          //增加触发使能次数
          l_i=0
          for l_i=0 to nAxesSum-1
            if bOpeEnabled==false
              // cst:nTO_DRVDISABLE=2
              if nCntDrvEnable[l_i]<250*cst:nTO_DRVDISABLE
                call cmdEnableOp(l_i)
              else
                sMsg="轴"+toString("",l_i+7)+"使能超时"
                popUpMsg(sMsg)
                logMsg(sMsg)
                bSysShut=true
                disablePower()
                return
              endIf
            endIf
            nCntDrvEnable[l_i]=nCntDrvEnable[l_i]+1
          endFor
        endIf
      else
        $setMaxPosErr(jZero)
        disablePower()
      endIf
    else
      bMemPower=false
      for l_i=0 to nAxesSum-1
        call cmdQuickStop(l_i)
      endFor
      //jDummy=$setMaxPosErr(jPosErrMax)
      // 设置驱动器位置反馈
      for l_i=0 to nAxesSum-1
        aioSet(aoIPPos[l_i],aioGet(aiPosFbk[l_i]))
      endFor
      $XsetDrvFbkPos(nDrvFbkPos)
    endIf
    delay(0)
  endWhile
end
